// Retrieves PLC Task information.
// [note] if not explicitly defined, the default task index is the task the function block is instatiated on. 
{attribute 'enable_dynamic_creation'}
{attribute 'no_explicit_call' := 'direct call for this function block is not allowed'}
FUNCTION_BLOCK FINAL FB_PlcTaskInformation IMPLEMENTS I_PlcTaskInformation
VAR
	_nTaskIndex : DINT;
END_VAR

// Task's ADS Port.
// [get] Returns the referenced task's ADS port.
PROPERTY AdsPort : Tc2_System.T_AmsPort
GET
AdsPort := TwinCAT_SystemInfoVarList._TaskInfo[THIS^._nTaskIndex].AdsPort;
END_GET
END_PROPERTY

// The task's cycle counter.
// [note] This refers to the actual system task and not to the task reference of the PLC project.
// [get] Returns the task's cycle counter.
PROPERTY CycleCount : UDINT
GET
CycleCount := TwinCAT_SystemInfoVarList._TaskInfo[THIS^._nTaskIndex].CycleCount;
END_GET
END_PROPERTY

// The cycle time of the task.
// [get] Returns the cycle time.
PROPERTY CycleTime : LTIME
GET
CycleTime := TO_LTIME(TwinCAT_SystemInfoVarList._TaskInfo[THIS^._nTaskIndex].CycleTime * 100);
END_GET
END_PROPERTY

// Indicates whether the cycle time has been exceeded.
// [get] Returns TRUE if the cycle time has been exceeded.
PROPERTY CycleTimeExceeded : BOOL
GET
CycleTimeExceeded := TwinCAT_SystemInfoVarList._TaskInfo[THIS^._nTaskIndex].CycleTimeExceeded;
END_GET
END_PROPERTY

{attribute 'hide'}
METHOD FB_init : BOOL
VAR_INPUT
	bInitRetains : BOOL; // if TRUE, the retain variables are initialized (warm start / cold start)
	bInCopyCode : BOOL;  // if TRUE, the instance afterwards gets moved into the copy code (online change)
END_VAR
VAR
	fbGetCurrentTaskIndex : Tc2_System.GETCURTASKINDEX;
END_VAR
fbGetCurrentTaskIndex(Index => THIS^._nTaskIndex);
END_METHOD

// Indicates if the origin of the current call is declared with the attribute 'TcCallAfterOutputUpdate'.
// [get] Returns TRUE if current call is declared with the attribute 'TcCallAfterOutputUpdate'.
PROPERTY HasCallAfterOutputUpdateAttribute : BOOL
GET
HasCallAfterOutputUpdateAttribute := TwinCAT_SystemInfoVarList._TaskInfo[THIS^._nTaskIndex].InCallAfterOutputUpdate;
END_GET
END_PROPERTY

// The index of the task.
// [get] Returns the index.
// [set] The index of the task to retrieve information from.
PROPERTY Index : DINT
GET
Index := THIS^._nTaskIndex;
END_GET
SET
THIS^._nTaskIndex := LIMIT(1, Index, F_SizeToDint(F_GetNumberOfPlcTasks()));
END_SET
END_PROPERTY

// Indicates if it is the first cycle of the task.
// [get] Returns TRUE if it is the first cycle.
PROPERTY IsFirstCycle : BOOL
GET
IsFirstCycle := TwinCAT_SystemInfoVarList._TaskInfo[THIS^._nTaskIndex].FirstCycle;
END_GET
END_PROPERTY

// Time the previous cycle took to complete execution.
// [get] Returns the last exection time.
PROPERTY LastCycleExecutionTime : LTIME
GET
LastCycleExecutionTime := TO_LTIME(TwinCAT_SystemInfoVarList._TaskInfo[THIS^._nTaskIndex].LastExecTime * 100);
END_GET
END_PROPERTY

// The name of the task.
// [get] Returns the task name.
PROPERTY Name : T_TaskNameString
GET
Name := TwinCAT_SystemInfoVarList._TaskInfo[THIS^._nTaskIndex].TaskName;
END_GET
END_PROPERTY

// The object ID of the task reference, from which the PLC program is called.
// [get] Returns the object ID.
PROPERTY ObjectId : OTCID
GET
ObjectId := TwinCAT_SystemInfoVarList._TaskInfo[THIS^._nTaskIndex].ObjId;
END_GET
END_PROPERTY

// The priority of the task.
// [get] Returns the priority.
PROPERTY Priority : UINT
GET
Priority := TwinCAT_SystemInfoVarList._TaskInfo[THIS^._nTaskIndex].Priority;
END_GET
END_PROPERTY

// Indicates whether the real-time time limit has been exceeded on a mixed core (Windows + real-time on one core).
// [get] Returns true if the real-time time limit has been exceeded.
PROPERTY RTTimeLimitExceeded : BOOL
GET
RTTimeLimitExceeded := TwinCAT_SystemInfoVarList._TaskInfo[THIS^._nTaskIndex].RTViolation;
END_GET
END_PROPERTY

END_FUNCTION_BLOCK

(* stored: Version 1.1.0.1
   POU FB_PlcTaskInformation: Id {d34eadf6-ab90-05ae-3a4a-66d09ffe82d0}, SpecialFunc None
   Property AdsPort: Id {8a378393-5fa1-0c1c-2120-627bd888d6fd}
   Get Get: Id {c5609cca-d812-0516-3514-cd22df14fb57}
   Property CycleCount: Id {606fb50b-63ff-0048-2a5f-f428ac78975d}
   Get Get: Id {07085d1f-6c35-0009-37d1-0134da5f6a25}
   Property CycleTime: Id {32ce03fc-9e1c-008c-125b-034c2b767fe4}
   Get Get: Id {74f59e60-fcb5-0978-234f-7bbf5ba522ee}
   Property CycleTimeExceeded: Id {1ec6bc54-7d90-0b68-292c-27dc0be3872b}
   Get Get: Id {f07f3c25-f257-07c7-2814-fc73d24522c4}
   Method FB_init: Id {6db93bfe-6854-0596-1361-e662b776c73e}
   Property HasCallAfterOutputUpdateAttribute: Id {a756ddea-8ab9-0e8a-1ed0-f540225211a0}
   Get Get: Id {0e79c0a8-916f-0e4b-3250-292d18ed8645}
   Property Index: Id {5cf7a19a-f68e-01e7-3a2b-04d52d95e5a4}
   Get Get: Id {fdddcd25-8bca-0dc0-0eae-0d4804e34446}
   Set Set: Id {d829f6a7-51a3-0f6d-2526-67a01b16bbb4}
   Property IsFirstCycle: Id {6d2dab56-79b0-0189-1c42-5566b3bf2887}
   Get Get: Id {f08221e4-aea8-0aac-1c55-2481a843e324}
   Property LastCycleExecutionTime: Id {31f57e75-8d6f-0bb7-38e9-979b01f4fe39}
   Get Get: Id {a857d344-5994-04c5-3480-ef236ba64db5}
   Property Name: Id {a18c1f0c-a7e5-0ac2-185e-e71c96dd403c}
   Get Get: Id {a998ca4d-ea89-05be-2fdc-7ee950909f21}
   Property ObjectId: Id {8cc46eee-8229-016e-2e83-6658635b532c}
   Get Get: Id {72b43474-349f-042c-12d9-4bea9f26e862}
   Property Priority: Id {2c545a4f-3316-0a69-2741-91d4e16d922b}
   Get Get: Id {59f08bf7-96f6-07e1-2712-e0272b96e0e7}
   Property RTTimeLimitExceeded: Id {6004deec-98d3-082a-172a-3285b148a293}
   Get Get: Id {81eea262-a5ec-0bf1-167d-ce782f8165de} *)
